TEXTLIST M_board_status
  0 = 'Offline'
  1 = 'Online'
   = ''
END_TEXTLIST

(* stored: Version 1.1.0.1, ProductVersion 3.1.4024.11
   TextList M_board_status: Id {d50dcf7a-023e-48ce-af4b-0cc3fae315e1} *)
